// TIA Portal V20 export
TYPE "LER_typeCmStatus"
// stored: Access Published
   STRUCT
      axisControl { ExternalWritable := 'False'} : Array[0..19] of "LBC_typeAxisControlNodeMonitoring";
      axis64PosControlNode { ExternalWritable := 'False'} : Array[0..19] of "LBC_typeAxis64PosControlNodeMonitoring";
      axis64PosConfig { ExternalWritable := 'False'} : Array[0..19] of "LBC_typeAxis64PosConfiguration";
      twoWayAct { ExternalWritable := 'False'} : Array[0..19] of "LBC_typeTwoWayActuatorControlNodeMonitoring";
      digitalSignal { ExternalWritable := 'False'} : Array[0..19] of "LBC_typeDigitalSignalControlNodeMonitoring";
      analogInput { ExternalWritable := 'False'} : Array[0..19] of "LBC_typeAnalogInputControlNodeMonitoring";
   END_STRUCT;
END_TYPE
